// Mitsubishi GX Works2 project: CCL   PLC: FX3U/FX3UC

PROGRAM MAIN
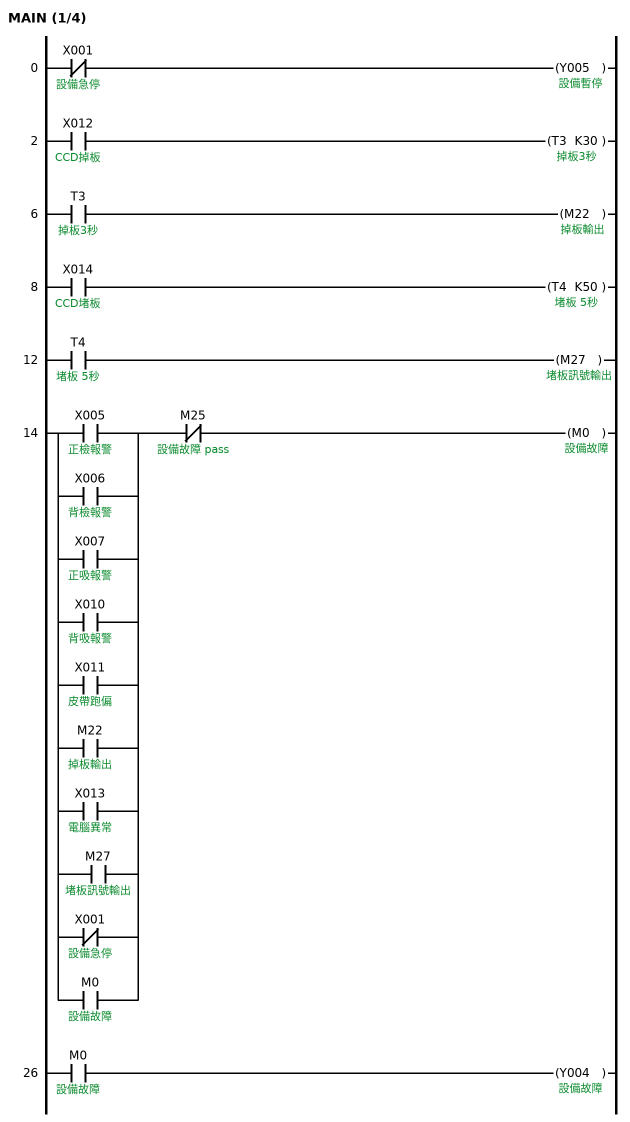
0     LDI     X001  ; 設備急停
      OUT     Y005  ; 設備暫停
2     LD      X012  ; CCD掉板
      OUT     T3 K30  ; 掉板3秒
6     LD      T3  ; 掉板3秒
      OUT     M22  ; 掉板輸出
8     LD      X014  ; CCD堵板
      OUT     T4 K50  ; 堵板 5秒
12    LD      T4  ; 堵板 5秒
      OUT     M27  ; 堵板訊號輸出
14    LD      X005  ; 正檢報警
      OR      X006  ; 背檢報警
      OR      X007  ; 正吸報警
      OR      X010  ; 背吸報警
      OR      X011  ; 皮帶跑偏
      OR      M22  ; 掉板輸出
      OR      X013  ; 電腦異常
      OR      M27  ; 堵板訊號輸出
      ORI     X001  ; 設備急停
      OR      M0  ; 設備故障
      ANI     M25  ; 設備故障 pass
      OUT     M0  ; 設備故障
26    LD      M0  ; 設備故障
      OUT     Y004  ; 設備故障
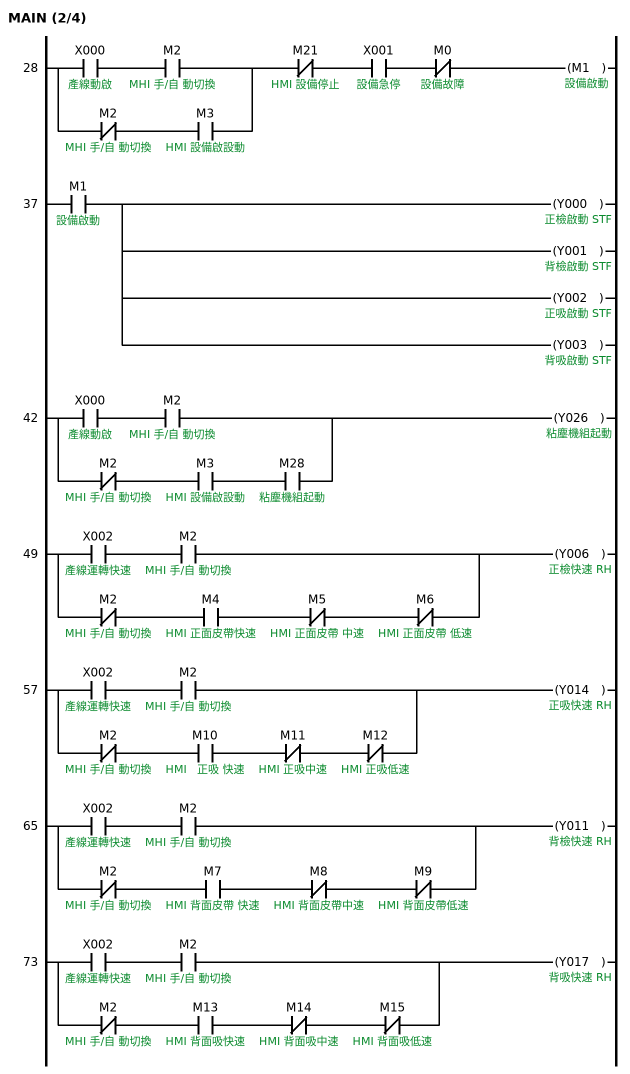
28    LD      X000  ; 產線動啟
      AND     M2  ; MHI 手/自 動切換
      LDI     M2  ; MHI 手/自 動切換
      AND     M3  ; HMI 設備啟設動
      ORB
      ANI     M21  ; HMI 設備停止
      AND     X001  ; 設備急停
      ANI     M0  ; 設備故障
      OUT     M1  ; 設備啟動
37    LD      M1  ; 設備啟動
      OUT     Y000  ; 正檢啟動 STF
      OUT     Y001  ; 背檢啟動 STF
      OUT     Y002  ; 正吸啟動 STF
      OUT     Y003  ; 背吸啟動 STF
42    LD      X000  ; 產線動啟
      AND     M2  ; MHI 手/自 動切換
      LDI     M2  ; MHI 手/自 動切換
      AND     M3  ; HMI 設備啟設動
      AND     M28  ; 粘塵機組起動
      ORB
      OUT     Y026  ; 粘塵機組起動
49    LD      X002  ; 產線運轉快速
      AND     M2  ; MHI 手/自 動切換
      LDI     M2  ; MHI 手/自 動切換
      AND     M4  ; HMI 正面皮帶快速
      ANI     M5  ; HMI 正面皮帶 中速
      ANI     M6  ; HMI 正面皮帶 低速
      ORB
      OUT     Y006  ; 正檢快速 RH
57    LD      X002  ; 產線運轉快速
      AND     M2  ; MHI 手/自 動切換
      LDI     M2  ; MHI 手/自 動切換
      AND     M10  ; HMI   正吸 快速
      ANI     M11  ; HMI 正吸中速
      ANI     M12  ; HMI 正吸低速
      ORB
      OUT     Y014  ; 正吸快速 RH
65    LD      X002  ; 產線運轉快速
      AND     M2  ; MHI 手/自 動切換
      LDI     M2  ; MHI 手/自 動切換
      AND     M7  ; HMI 背面皮帶 快速
      ANI     M8  ; HMI 背面皮帶中速
      ANI     M9  ; HMI 背面皮帶低速
      ORB
      OUT     Y011  ; 背檢快速 RH
73    LD      X002  ; 產線運轉快速
      AND     M2  ; MHI 手/自 動切換
      LDI     M2  ; MHI 手/自 動切換
      AND     M13  ; HMI 背面吸快速
      ANI     M14  ; HMI 背面吸中速
      ANI     M15  ; HMI 背面吸低速
      ORB
      OUT     Y017  ; 背吸快速 RH
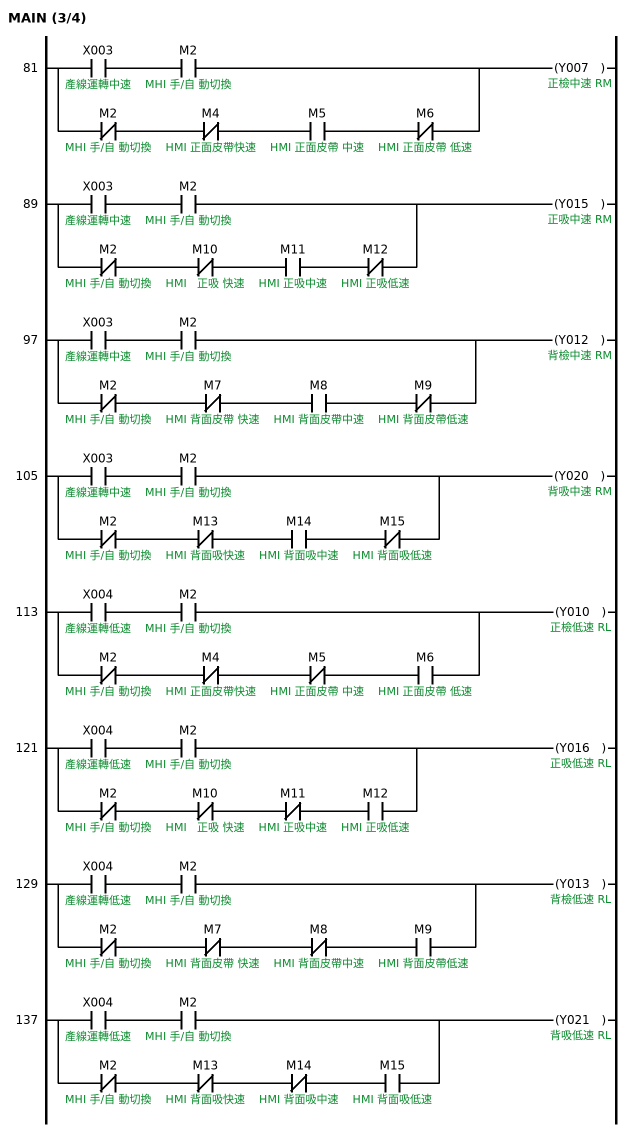
81    LD      X003  ; 產線運轉中速
      AND     M2  ; MHI 手/自 動切換
      LDI     M2  ; MHI 手/自 動切換
      ANI     M4  ; HMI 正面皮帶快速
      AND     M5  ; HMI 正面皮帶 中速
      ANI     M6  ; HMI 正面皮帶 低速
      ORB
      OUT     Y007  ; 正檢中速 RM
89    LD      X003  ; 產線運轉中速
      AND     M2  ; MHI 手/自 動切換
      LDI     M2  ; MHI 手/自 動切換
      ANI     M10  ; HMI   正吸 快速
      AND     M11  ; HMI 正吸中速
      ANI     M12  ; HMI 正吸低速
      ORB
      OUT     Y015  ; 正吸中速 RM
97    LD      X003  ; 產線運轉中速
      AND     M2  ; MHI 手/自 動切換
      LDI     M2  ; MHI 手/自 動切換
      ANI     M7  ; HMI 背面皮帶 快速
      AND     M8  ; HMI 背面皮帶中速
      ANI     M9  ; HMI 背面皮帶低速
      ORB
      OUT     Y012  ; 背檢中速 RM
105   LD      X003  ; 產線運轉中速
      AND     M2  ; MHI 手/自 動切換
      LDI     M2  ; MHI 手/自 動切換
      ANI     M13  ; HMI 背面吸快速
      AND     M14  ; HMI 背面吸中速
      ANI     M15  ; HMI 背面吸低速
      ORB
      OUT     Y020  ; 背吸中速 RM
113   LD      X004  ; 產線運轉低速
      AND     M2  ; MHI 手/自 動切換
      LDI     M2  ; MHI 手/自 動切換
      ANI     M4  ; HMI 正面皮帶快速
      ANI     M5  ; HMI 正面皮帶 中速
      AND     M6  ; HMI 正面皮帶 低速
      ORB
      OUT     Y010  ; 正檢低速 RL
121   LD      X004  ; 產線運轉低速
      AND     M2  ; MHI 手/自 動切換
      LDI     M2  ; MHI 手/自 動切換
      ANI     M10  ; HMI   正吸 快速
      ANI     M11  ; HMI 正吸中速
      AND     M12  ; HMI 正吸低速
      ORB
      OUT     Y016  ; 正吸低速 RL
129   LD      X004  ; 產線運轉低速
      AND     M2  ; MHI 手/自 動切換
      LDI     M2  ; MHI 手/自 動切換
      ANI     M7  ; HMI 背面皮帶 快速
      ANI     M8  ; HMI 背面皮帶中速
      AND     M9  ; HMI 背面皮帶低速
      ORB
      OUT     Y013  ; 背檢低速 RL
137   LD      X004  ; 產線運轉低速
      AND     M2  ; MHI 手/自 動切換
      LDI     M2  ; MHI 手/自 動切換
      ANI     M13  ; HMI 背面吸快速
      ANI     M14  ; HMI 背面吸中速
      AND     M15  ; HMI 背面吸低速
      ORB
      OUT     Y021  ; 背吸低速 RL
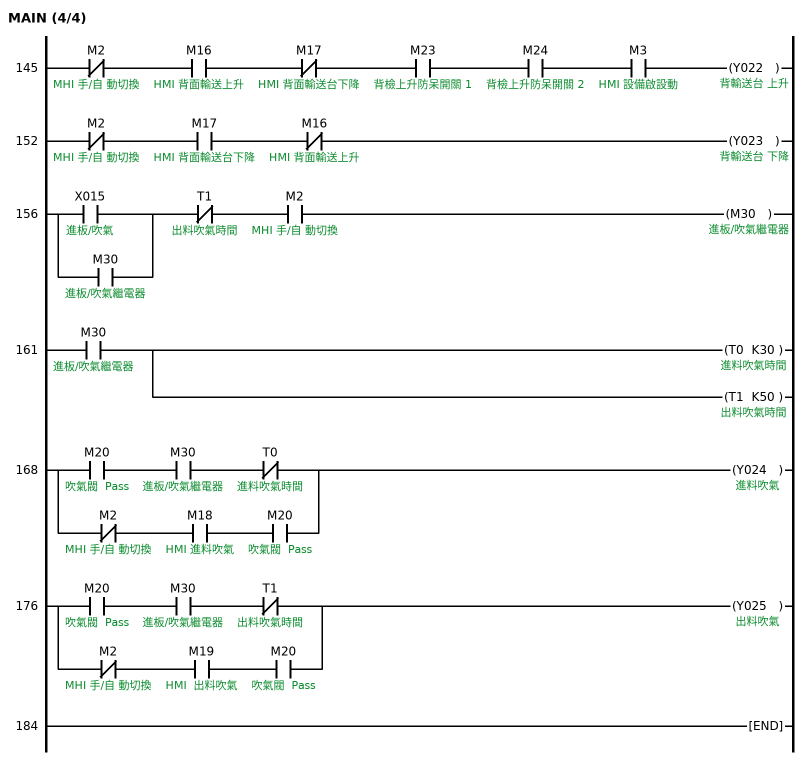
145   LDI     M2  ; MHI 手/自 動切換
      AND     M16  ; HMI 背面輸送上升
      ANI     M17  ; HMI 背面輸送台下降
      AND     M23  ; 背檢上升防呆開關 1
      AND     M24  ; 背檢上升防呆開關 2
      AND     M3  ; HMI 設備啟設動
      OUT     Y022  ; 背輸送台 上升
152   LDI     M2  ; MHI 手/自 動切換
      AND     M17  ; HMI 背面輸送台下降
      ANI     M16  ; HMI 背面輸送上升
      OUT     Y023  ; 背輸送台 下降
156   LD      X015  ; 進板/吹氣
      OR      M30  ; 進板/吹氣繼電器
      ANI     T1  ; 出料吹氣時間
      AND     M2  ; MHI 手/自 動切換
      OUT     M30  ; 進板/吹氣繼電器
161   LD      M30  ; 進板/吹氣繼電器
      OUT     T0 K30  ; 進料吹氣時間
      OUT     T1 K50  ; 出料吹氣時間
168   LD      M20  ; 吹氣閥  Pass
      AND     M30  ; 進板/吹氣繼電器
      ANI     T0  ; 進料吹氣時間
      LDI     M2  ; MHI 手/自 動切換
      AND     M18  ; HMI 進料吹氣
      AND     M20  ; 吹氣閥  Pass
      ORB
      OUT     Y024  ; 進料吹氣
176   LD      M20  ; 吹氣閥  Pass
      AND     M30  ; 進板/吹氣繼電器
      ANI     T1  ; 出料吹氣時間
      LDI     M2  ; MHI 手/自 動切換
      AND     M19  ; HMI  出料吹氣
      AND     M20  ; 吹氣閥  Pass
      ORB
      OUT     Y025  ; 出料吹氣
184   END
END_PROGRAM

// device comments not shown above
M26  ; 吸風自動/旋鈕切換
D0  ; HMI 吹氣秒數
D3  ; PLC 吹氣輸出秒數
